Yaskawa INFORM job: 50_smooth.JBI

/JOB
//NAME AAA
//POS
///NPOS 4,0,0,0,0,0
///TOOL 10
///POSTYPE PULSE
///PULSE
C00000=31970,-841,-7031,9752,-64737,-11903
C00001=31970,-841,-7031,9752,-64737,-11903
C00002=-26929,-6371,-25778,-51792,-72912,10976
C00003=-58721,56844,404,-80660,-106680,14278
//INST
///DATE 2023/04/04 11:55
///ATTR SC,RW
///GROUP1 RB1
NOP
MOVJ C00000 VJ=5.0
TIMER T=1.00
MOVJ C00001 VJ=1.0
TIMER T=0.10
MOVL C00002 V=50.0 PL=1
MOVL C00003 V=50.0 PL=1
END
